TYPE
    ST_MoveStates : STRUCT
        Idle    : UDINT;
        Pick    : UDINT;
        Hold    : UDINT;
        Clear   : UDINT;
        Drop    : UDINT;
        Grab    : UDINT;
        Release : UDINT;
    END_STRUCT
END_TYPE

(* stored: Version 1.1.0.1
   DUT ST_MoveStates: Id {29f68f7c-f85f-4dc1-824c-82553d0bc5c5} *)
